//		IF(NOT simpleCommand.xError AND simpleCommand.xDone)THEN
//			iterateAndUpdateStatus.isInit := TRUE;
//			error := CRT_NO_ERROR;
//		END_IF
	CRT_CLOSE_COM_STATE:
		state := CRT_RESET_STATE;
		IF b_crt_close_enable THEN
			IF portOpened THEN
				crtClose(xExecute:=TRUE, hCom := openedHCom);
				IF crtClose.xError THEN
				   portOpened := FALSE;
				   crtClose.xExecute := FALSE;
				   state := CRT_INIT_STATE;
				   error := CRT_OPEN_ERROR;
				END_IF;
				IF crtClose.xDone THEN
					portOpened := FALSE;
				   crtClose.xExecute := FALSE;
				   state := CRT_INIT_STATE;
				END_IF;
			ELSE
				   state := CRT_INIT_STATE;
			END_IF
			
		END_IF
		
	
	CRT_STATUS_REQUEST_STATE:	
		simpleCommand(xExecute:=TRUE, hCom := openedHCom, xCommandDataSize:=0, xCommand:= CRT_STATUS_REQUEST_COMMAND , xCommandDataSize:=0);
		IF simpleCommand.xDone THEN
			newCardState := crtDecodeCardState(iST0:=simpleCommand.xST0, iST1:=simpleCommand.xST1);
			locked := (simpleCommand.xST1 = 16#30); 
			state := CRT_STATUS_REQUEST_STATE;
			waitTimer(IN:= TRUE, PT := POLL_DELAY);
			
		END_IF
		

		IF simpleCommand.xError THEN    
			newCardState := CRT_CARD_UNDEFINED;
			IF simpleCommand.xTimeout THEN
				state := CRT_CLOSE_COM_STATE;
				waitTimer(IN:= TRUE, PT := POLL_DELAY);
			ELSE
				//state := CRT_STATUS_REQUEST_STATE;
				state := CRT_CLOSE_COM_STATE;
				waitTimer(IN:= TRUE, PT := POLL_DELAY);
			END_IF
		END_IF	
	CRT_RF_CARD_RESET:
		simpleCommand(xExecute:=TRUE, hCom := openedHCom,  xCommand:= CRT_RF_CARD_RESET_COMMAND , 
				     xCommandDataSize:=UINT_TO_BYTE(SIZEOF(CRT_RF_CARD_RESET_COMMAND_DATA)), xCommandData := ADR (CRT_RF_CARD_RESET_COMMAND_DATA)) ;
		IF simpleCommand.xDone THEN
			//newCardState := crtDecodeCardState(iST0:=simpleCommand.xST0, iST1:=simpleCommand.xST1);
			newCardState :=CRT_RF_CARD_INSIDE;
			state := CRT_STATUS_REQUEST_STATE;
			waitTimer(IN:= TRUE, PT := POLL_DELAY);
			cardIdLen := simpleCommand.xOutputData[3];
			MEM.MemMove(pSource:=simpleCommand.xOutputData + 4, pDestination:=ADR(cardId), uiNumberOfBytes := MIN(cardIdLen, SIZEOF(cardId)));
			
		END_IF
		

		IF simpleCommand.xError THEN    
			newCardState := CRT_CARD_UNDEFINED;
			IF simpleCommand.xTimeout THEN
				//state := CRT_RESET_STATE;
				state := CRT_CLOSE_COM_STATE;
				waitTimer(IN:= TRUE, PT := POLL_DELAY);
			ELSE
				//state := CRT_STATUS_REQUEST_STATE;
				state := CRT_CLOSE_COM_STATE;
				waitTimer(IN:= TRUE, PT := POLL_DELAY);
			END_IF
		END_IF	

	CRT_LOCK:
		simpleCommand(xExecute:=TRUE, hCom := openedHCom, xCommandDataSize:=0, xCommand:= CRT_LATCH_LOCK_COMMAND , xCommandDataSize:=0);
		IF simpleCommand.xDone THEN
			newCardState := crtDecodeCardState(iST0:=simpleCommand.xST0, iST1:=simpleCommand.xST1);
			locked := (simpleCommand.xST1 = 16#30); 
			state := CRT_STATUS_REQUEST_STATE;
			waitTimer(IN:= TRUE, PT := POLL_DELAY);
			
		END_IF

		IF simpleCommand.xError THEN    
			newCardState := CRT_CARD_UNDEFINED;
			IF simpleCommand.xTimeout THEN
				//state := CRT_RESET_STATE;
				state := CRT_CLOSE_COM_STATE;
				waitTimer(IN:= TRUE, PT := POLL_DELAY);
			ELSE
				//state := CRT_STATUS_REQUEST_STATE;
				state := CRT_CLOSE_COM_STATE;
				waitTimer(IN:= TRUE, PT := POLL_DELAY);
			END_IF
		END_IF		

	CRT_RELEASE:
		simpleCommand(xExecute:=TRUE, hCom := openedHCom, xCommandDataSize:=0, xCommand:= CRT_LATCH_RELEASE_COMMAND , xCommandDataSize:=0);
		IF simpleCommand.xDone THEN
			newCardState := crtDecodeCardState(iST0:=simpleCommand.xST0, iST1:=simpleCommand.xST1);
			locked := (simpleCommand.xST1 = 16#30); 
			state := CRT_STATUS_REQUEST_STATE;
			waitTimer(IN:= TRUE, PT := POLL_DELAY);
			
		END_IF

		IF simpleCommand.xError THEN    
			newCardState := CRT_CARD_UNDEFINED;
			IF simpleCommand.xTimeout THEN
				//state := CRT_RESET_STATE;
				state := CRT_CLOSE_COM_STATE;
				waitTimer(IN:= TRUE, PT := POLL_DELAY);
			ELSE
				//state := CRT_STATUS_REQUEST_STATE;
				state := CRT_CLOSE_COM_STATE;
				waitTimer(IN:= TRUE, PT := POLL_DELAY);
			END_IF
		END_IF					
	
		
    CRT_FATAL_ERROR:
		state := CRT_CLOSE_COM_STATE;
	
//	CRT_DONE:  //all work is done, free resources
//		crtOpen(xExecute := FALSE);
//		state := CRT_DO_NOTHING;
//						
//	CRT_DO_NOTHING:
END_CASE

IF newCardState = CRT_CARD_INSIDE AND lastCardState = CRT_RF_CARD_INSIDE THEN 
	newCardState := CRT_RF_CARD_INSIDE;
END_IF

IF newCardState = CRT_CARD_INSIDE AND lastCardState <> CRT_CARD_INSIDE THEN
	//moment of inserting card
	state := CRT_RF_CARD_RESET;
	waitTimer(IN:= TRUE, PT := POLL_DELAY);
ELSIF newCardState <> CRT_CARD_INSIDE AND newCardState <> CRT_RF_CARD_INSIDE THEN
	cardIdLen :=0; //reset card id
	
END_IF		
lastCardState := newCardState;

iterateAndUpdateStatus.cardState := newCardState;
iterateAndUpdateStatus.busy := simpleCommand.xExecute OR NOT crtOpen.xDone;
//iterateAndUpdateStatus.busy := (simpleCommand.xExecute AND NOT simpleCommand.xDone) OR NOT crtOpen.xDone;
iterateAndUpdateStatus.locked := locked;
iterateAndUpdateStatus.error := error;
END_METHOD

METHOD latchLock
//very stupid
IF  state <> CRT_FATAL_ERROR AND state <> CRT_DONE AND state <> CRT_RESET_STATE AND state<>CRT_DO_NOTHING THEN
	state:= CRT_LOCK;

END_IF
END_METHOD

METHOD latchRelease
IF  state <> CRT_FATAL_ERROR AND state <> CRT_DONE AND state <> CRT_RESET_STATE AND state<>CRT_DO_NOTHING THEN
	state:= CRT_RELEASE;

END_IF
END_METHOD

END_FUNCTION_BLOCK

// CompWin/AppTerminalPost/DevCard/crtSimpleCommand
///command 
FUNCTION_BLOCK crtSimpleCommand
VAR CONSTANT
	STATE_INITIAL: BYTE := 0;
	STATE_WAIT_ACK: BYTE := 1;
	STATE_FATAL_ERROR: BYTE := 3;
	STATE_WAIT_RESPONSE: BYTE := 4;
	STATE_SEND_ACK: BYTE := 5;
	///minimal answer
	COMMAND_MINIMAL_ANSWER_SIZE: BYTE := 9;
	///maximum size of command data 
	COMMAND_DATA_SIZE_MAX: BYTE := 5;
	///maximum size of response 
	RESPONSE_DATA_SIZE_MAX: BYTE := 255;
	COMMAND_DATA_OFFSET: BYTE := 6;
	RESPONSE_DATA_OFFSET: BYTE := 8;
	ACK: BYTE := 16#6;
	///? 
	TIMEOUT: TIME := TIME#2s0ms;
END_VAR
VAR_INPUT
	hCom: CAA.HANDLE;
	xExecute: BOOL := FALSE;
	///device address
	xDestinationId: BYTE := 2;
	///master address, default = 1;
	xSourceId: BYTE := 1;
	xCommand: crtParametrizedCommand;
	xCommandData: POINTER TO BYTE;
	xCommandDataSize: BYTE := 0;
END_VAR
VAR_OUTPUT
	xDone: BOOL := FALSE;
	xError: BOOL := FALSE;
	xTimeout: BOOL := FALSE;
	///status characters
	xST0: BYTE;
	xST1: BYTE;
	///error codes
	xE0: BYTE;
	xE1: BYTE;
	xOutputData: POINTER TO BYTE := ((ADR(readBuffer) + RESPONSE_DATA_OFFSET) + 1);
	xOutputDataSize: BYTE;
END_VAR
VAR
	///buffer for command
	commandBuffer: ARRAY[0..(((2 + 3) + COMMAND_DATA_SIZE_MAX) + 2)] OF BYTE;
	///size enough for ack and answer
	readBuffer: ARRAY[0..(((3 + 3) + RESPONSE_DATA_SIZE_MAX) + 2)] OF BYTE;
	///timeout timer (timeout value - ????)
	waitingACKtimeout: TON;
	localState: BYTE := STATE_INITIAL;
	crtCOMWrite: COM.Write;
	crtCOMRead: COM.Read;
	bufferReaded: CAA.SIZE := 0;
	bufferFullLen: BYTE := 5;
	///full answer size with echo
	fullAnswerSize: BYTE;
	errorExecuting: BOOL;
	commandCode: INT;
	bcc: BYTE;
END_VAR

CASE localState OF 
	STATE_INITIAL:
		IF xExecute THEN
			xDone := FALSE;
			xError := FALSE;
			xTimeout := FALSE;
			IF NOT crtCOMWrite.xExecute THEN //at first time fill buffer
				bufferFullLen := 3 + 3 + xCommandDataSize + 2;  
				commandBuffer[0] := 16#F2;    //header 1
				commandBuffer[1] := 0;    //data len msb
				commandBuffer[2] := 3 + xCommandDataSize; //data len lsb
				commandBuffer[3] := 16#43;
				commandBuffer[4] := xCommand.CM; 		   //CM (command character)
				commandBuffer[5] := xCommand.PM;  //PM (parameter character)
				xOutputDataSize := 0;
				IF xCommandDataSize > 0 THEN
					MEM.MemMove(pSource := xCommandData, pDestination := ADR(commandBuffer) + COMMAND_DATA_OFFSET, uiNumberOfBytes := xCommandDataSize);
				END_IF;
				commandBuffer[6 + xCommandDataSize]:= 3; //don't know, what is it
				commandBuffer[7 + xCommandDataSize] := crtBCC(iCommandBuffer := ADR(commandBuffer) , iCommandBufferSize := bufferFullLen);
				xE0 :=0;
				xE1 :=0;
				errorExecuting :=FALSE;

			END_IF
			crtCOMWrite(xExecute := TRUE,hCom:= hCom, pBuffer:= ADR(commandBuffer), szSize:= bufferFullLen);
			IF crtCOMWrite.xError THEN
				xError := TRUE;
				xExecute := FALSE;
				xCommandDataSize :=0;
				localState := STATE_INITIAL;
				crtCOMWrite(xExecute := FALSE);
				RETURN;
			END_IF
		
			// if the writing process is completed the reading process can be started
			IF crtCOMWrite.xDone THEN
				localState := STATE_WAIT_RESPONSE;
				bufferReaded := 0;
				xCommandDataSize :=0;
				crtCOMWrite(xExecute := FALSE);
				fullAnswerSize := COMMAND_MINIMAL_ANSWER_SIZE; //wait for ack + response
				errorExecuting := FALSE;
				waitingACKtimeout(IN:=FALSE); 
				waitingACKtimeout(IN:=TRUE, PT:=TIMEOUT);  //timeout value ?
			END_IF			
		END_IF
	//waiting response and ack
	STATE_WAIT_RESPONSE:
		waitingACKtimeout(IN:=TRUE, PT:=TIMEOUT);  //timeout value ?
		IF waitingACKTimeout.Q THEN  //timeout is over..
			xError := TRUE;
			xExecute := FALSE;
			xTimeout := TRUE;
			localState := STATE_INITIAL;
			crtCOMRead(xExecute := FALSE);
		ELSE
			crtCOMRead(xExecute := FALSE);
			crtCOMRead(xExecute := TRUE,hCom:= hCom, pBuffer:= ADR(readBuffer) + bufferReaded, szBuffer:= SIZEOF(readBuffer) - bufferReaded);
			IF crtCOMRead.xError THEN
				xError := TRUE;
				xExecute := FALSE;
				crtCOMRead(xExecute := FALSE);
				localState := STATE_INITIAL;
			END_IF
			//After completion the size of the written bytes are saved
			IF 	crtCOMRead.xDone THEN
				bufferReaded := bufferReaded + crtCOMRead.szSize;
				//if first byte not ack-errir
				IF bufferReaded >=1 AND readBuffer[0]<> ACK THEN
					xError := TRUE;
					xExecute := FALSE;
					crtCOMRead(xExecute := FALSE);
					localState := STATE_INITIAL;
					RETURN;
				END_IF 
				IF bufferReaded >= fullAnswerSize THEN  //try to recognize command
					crtCOMRead(xExecute := FALSE);
					//ALL OK
					IF (readBuffer[1] = 16#F2 AND readBuffer[5]= xCommand.CM AND readBuffer[6]= xCommand.PM ) THEN  //receive response
						localState := STATE_WAIT_RESPONSE;
						fullAnswerSize := readBuffer[3] + 5 + 1; //extract response data size from readbuffer (with ACK FIRST BYTE)
						IF (bufferReaded >= fullAnswerSize ) THEN
							crtCOMRead(xExecute := FALSE);
							bcc := crtBCC(iCommandBuffer := ADR(readBuffer) +1, iCommandBufferSize := fullAnswerSize-1);
							IF bcc = readBuffer[fullAnswerSize - 1] AND readBuffer[4] = 16#50 THEN  //ordinary response, all ok
								xST1:= readBuffer[7];
								xST0:= readBuffer[8];
								xOutputDataSize := readBuffer[3] - 3;
								localState := STATE_SEND_ACK;
							ELSIF bcc = readBuffer[fullAnswerSize - 1] AND readBuffer[4] = 16#4E THEN //irregular response 								
								xE1:=readBuffer[7];
								xE0:=readBuffer[8];
								xOutputDataSize := readBuffer[3] - 3;
								errorExecuting := TRUE;
								localState := STATE_SEND_ACK;
							ELSE
								xError := TRUE;
								xExecute := FALSE;
								localState := STATE_INITIAL;
							END_IF
						END_IF
					ELSE
						xError := TRUE;
						xExecute := FALSE;
						localState := STATE_INITIAL;
					END_IF
				END_IF

			END_IF			
		END_IF
	STATE_SEND_ACK:
		commandBuffer[0] := 16#06; //ACK 
		crtCOMWrite(xExecute := TRUE,hCom:= hCom, pBuffer:= ADR(commandBuffer), szSize:= 1); //send ack
		IF crtCOMWrite.xError OR crtCOMWrite.xDone  THEN
				xExecute := FALSE;
				xError := errorExecuting;
				xDone := NOT (xError);
				
				xCommandDataSize :=0;
				localState := STATE_INITIAL;
				crtCOMWrite(xExecute := FALSE);
				RETURN;
		END_IF
		
		
		
END_CASE

END_FUNCTION_BLOCK

// CompWin/AppTerminalPost/DevCard/crtBCC
///calculate BCC (exclusive-or-verify) for buffer; receive full command buffer
FUNCTION crtBCC : BYTE
VAR_INPUT
	iCommandBuffer: POINTER TO BYTE;
	iCommandBufferSize: WORD;
END_VAR
VAR
	i: WORD;
END_VAR

crtBCC := 0;
FOR i := 0 TO iCommandBufferSize - 2 DO
	crtBCC := crtBCC XOR iCommandBuffer[i];
END_FOR

END_FUNCTION

// CompWin/AppTerminalPost/DevCard/crtDecodeCardState
///process ST0 and ST1 status command output
FUNCTION crtDecodeCardState : CRT_CARD_STATE
VAR_INPUT
	iST0: BYTE;
	iST1: BYTE;
END_VAR

crtDecodeCardState := CRT_CARD_UNDEFINED;
IF (iST0 =16#30 OR iST0 = 16#31) THEN
	crtDecodeCardState := CRT_NO_CARD;
ELSIF iST0 = 16#32 THEN
	crtDecodeCardState := CRT_CARD_INSIDE;
END_IF

END_FUNCTION

// CompWin/AppTerminalPost/StdLogger
FUNCTION_BLOCK StdLogger
VAR_INPUT
	sCmpName  : STRING;
END_VAR
VAR_OUTPUT
END_VAR
VAR
	udiCmpId : UDINT;
	udiCmpVersion : UDINT;
	vendorId : UDINT := 16#11110000;
	cmpId : UDINT := 16#0123;
	hCmp : RTS_IEC_HANDLE;
	hStdLogger : RTS_IEC_HANDLE;
	Result : RTS_IEC_RESULT;
	c: INT := 0;	
END_VAR

udiCmpId := vendorId OR Component_Manager.ComponentID.CMPID_IecCode OR cmpId;
udiCmpVersion := 16#03050000;
//sCmpName := 'CashCode';
//hCmp := CMAddComponent(sCmpName, udiCmpId, udiCmpVersion, ADR(Result)); 
hCmp := CMAddComponent('CashCode', udiCmpId, udiCmpVersion, ADR(Result));

METHOD AddLogEntry : BOOL
VAR_INPUT
	udiClassId : UDINT;
	sText : WSTRING;
END_VAR
VAR
	str: STRING;
	udiErrorId : UDINT := Errors.ERR_FAILED;
	udiInfoId : UDINT := 0;
END_VAR
AddLogEntry := FALSE;
str := WSTRING_TO_STRING(sText);
IF (LogAdd2(hStdLogger, udiCmpId, udiClassId, udiErrorId, udiInfoId, str) = Errors.ERR_OK) THEN
	AddLogEntry := TRUE;
END_IF;
END_METHOD

METHOD debug
VAR_INPUT
	msg: WSTRING;
END_VAR
AddLogEntry(CmpLog.LogClass.LOG_DEBUG, msg);
END_METHOD

METHOD error
VAR_INPUT
	msg: WSTRING;
END_VAR
AddLogEntry(CmpLog.LogClass.LOG_ERROR, msg);
END_METHOD

METHOD FB_Exit : BOOL
VAR_INPUT
	bInCopyCode : BOOL;  // if TRUE, the instance afterwards gets moved into the copy code (online change)	
END_VAR
CMRemoveComponent(hCmp);
FB_exit := TRUE;
END_METHOD

METHOD FB_Init : BOOL
VAR_INPUT
	bInitRetains : BOOL; // if TRUE, the retain variables are initialized (warm start / cold start)
	bInCopyCode : BOOL;  // if TRUE, the instance afterwards gets moved into the copy code (online change)	
END_VAR
c := c + 1;

hStdLogger := LogOpen('PlcLog', 0);
FB_Init := TRUE;
END_METHOD

METHOD info
VAR_INPUT
	msg: WSTRING;
END_VAR
AddLogEntry(CmpLog.LogClass.LOG_INFO, msg);
END_METHOD

METHOD warn
VAR_INPUT
	msg: WSTRING;
END_VAR
AddLogEntry(CmpLog.LogClass.LOG_WARNING, msg);
END_METHOD

END_FUNCTION_BLOCK

// CompWin/AppTerminalPost/Post/SafePrg
PROGRAM SafePrg

// сохранить retain в файл
IF(RetainManager.Init)THEN
//	RetainManager(ForceRestore := FALSE, ForceSave := TRUE, ForceBalance := FALSE);
	RetainManager(ForceRestore := FALSE, ForceSave := FALSE, ForceBalance := FALSE);
END_IF

END_PROGRAM

// CompWin/AppTerminalPost/Traffic/DataToSpk
PROGRAM DataToSpk
VAR
	_activeButton : INT;
END_VAR

// номер поста
//go_postNumber := PLC_PRG.post.Number;
// выбранная функция
_activeButton := DeviceButtons.GetActiveButton();// PLC_PRG.post.Mode;
// для режимов не_мойки не передавать ничего в Контроллер
//IF(PLC_PRG.post.Mode = EnumMode.CASHCOLLECT)THEN
IF(NOT PLC_PRG.post.IsReadyToWash())THEN
	spk_data.go_postFunction := EnumButton.NONE;
ELSE
	spk_data.go_postFunction := _activeButton;
END_IF


// изменение для замены местами пены и шампуня
IF(spk_data.go_postFunction = 2)THEN
	spk_data.go_postFunction := 3;
ELSIF(spk_data.go_postFunction = 3)THEN
	spk_data.go_postFunction := 2;
END_IF

// баланс поста
spk_data.go_postCounterFund := REAL_TO_INT(PLC_PRG.post.CounterFund);

// счётчики банкнот
SPK_DATA.counterBanknote10 := DeviceBanknote.GetCounterBanknote(10);
SPK_DATA.counterBanknote50 := DeviceBanknote.GetCounterBanknote(50);
SPK_DATA.counterBanknote100 := DeviceBanknote.GetCounterBanknote(100);
SPK_DATA.counterBanknote500 := DeviceBanknote.GetCounterBanknote(500);
SPK_DATA.counterBanknote1000 := DeviceBanknote.GetCounterBanknote(1000);
SPK_DATA.counterBanknote5000 := DeviceBanknote.GetCounterBanknote(5000);

// счётчики монет
SPK_DATA.counterCoin := DeviceCoin.GetCounterCoin(0);
SPK_DATA.counterCoin1 := DeviceCoin.GetCounterCoin(1);
SPK_DATA.counterCoin2 := DeviceCoin.GetCounterCoin(2);
SPK_DATA.counterCoin5 := DeviceCoin.GetCounterCoin(5);
SPK_DATA.counterCoin10 := DeviceCoin.GetCounterCoin(10);

SPK_DATA.fundFromCollect := PLC_PRG.post.GeFundFromCollect();
SPK_DATA.fundTotal := PLC_PRG.post.GetFundTotal();

// сообщения
SPK_DATA.messageInCash := PLC_PRG.post.GetMessageInCash();
SPK_DATA.messageFunc := PLC_PRG.post.GetMessageFunc();
SPK_DATA.messageCollect := PLC_PRG.post.GetMessageCollect();
SPK_DATA.messageTotal := PLC_PRG.post.GetMessageTotal();

// счетчик для контроля связи и работы терминала
spk_data.go_counter := spk_data.go_counter + 1;

// показать текущие тарифы мойки
SPK_DATA.currentRates[0] := PersistentVars.rates[0];
SPK_DATA.currentRates[1] := PersistentVars.rates[1];
SPK_DATA.currentRates[2] := PersistentVars.rates[2];
SPK_DATA.currentRates[3] := PersistentVars.rates[3];
SPK_DATA.currentRates[4] := PersistentVars.rates[4];
SPK_DATA.currentRates[5] := PersistentVars.rates[5];
SPK_DATA.currentRates[6] := PersistentVars.rates[6];
SPK_DATA.currentRates[7] := PersistentVars.rates[7];
SPK_DATA.currentRates[8] := PersistentVars.rates[8];


// Флаги купюрника
SPK_DATA.cashcodeStatus := DeviceBanknote.cashcodeStatus;
SPK_DATA.cashcodeError := DeviceBanknote.cashcodeError;
SPK_DATA.casetteDropped := DeviceBanknote.IsCasetteDropped();
SPK_DATA.banknoteJammed := DeviceBanknote.IsBanknoteJammed();

// Флаги блокировки дверей
// 1 - замок закрыт; 0 - замок открыт
IF(PLC_PRG.post.Locks[EnumLock.LOCK_TOP])THEN
	SPK_DATA.lockTop := 1;
ELSE
	SPK_DATA.lockTop := 0;
END_IF

// состояние среднего замка
IF(PLC_PRG.post.Locks[EnumLock.LOCK_MID])THEN
	SPK_DATA.lockMid := 1;
ELSE
	SPK_DATA.lockMid := 0;
END_IF

// текущие паузы режимов
SPK_DATA.currentPauseActiveClean := TIME_TO_WORD(PLC_PRG.post.GetPauseActiveClean() / 1000);
SPK_DATA.currentPauseFoam := TIME_TO_WORD(PLC_PRG.post.GetPauseFoam() / 1000);
SPK_DATA.currentPauseShampoo := TIME_TO_WORD(PLC_PRG.post.GetPauseShampoo() / 1000);

END_PROGRAM

// CompWin/AppTerminalPost/Traffic/DataToUI
PROGRAM DataToUI
VAR
END_VAR

// номер поста
NVL2UI.postNumber := PLC_PRG.post.Number;
	
// Состояние терминала: ожидание, функции, окончание мойки, уборка, инкассация, пополнение баланса оператором
NVL2UI.postMode := PLC_PRG.post.Mode;
IF(PLC_PRG.post.ActiveCardType = EnumCardType.CLEANUP)THEN
	NVL2UI.postMode := EnumMode.CLEANUP;
//ELSIF(PLC_PRG.post.ActiveCardType = EnumCardType.CASHCOLLECT)THEN
//	
END_IF

// Для REAL отбросываю дробную часть DINT_TO_INT(TRUNC(real));
// REAL_TO_WORD(real);	// округление до ближайшего целого
// баланс
NVL2UI.postCounterFund := DINT_TO_INT(TRUNC(PLC_PRG.post.CounterFund));

// тип карты
NVL2UI.cardType := PLC_PRG.post.ActiveCardType;

	
// нажатая кнопка
NVL2UI.buttonActive := DeviceButtons.GetActiveButton();
// изменение для замены местами пены и шампуня
IF(NVL2UI.buttonActive = 2)THEN
	NVL2UI.buttonActive := 3;
ELSIF(NVL2UI.buttonActive = 3)THEN
	NVL2UI.buttonActive := 2;
END_IF
		
// сумма внесения
NVL2UI.amountReceived := WORD_TO_INT(PLC_PRG.post.Received);
	
IF(PLC_PRG.post.FinCostSummary <> '')THEN	
	// внесено за мойку
	//NVL2UI.paidWash := PLC_PRG.post.InCash;
	// стоимость оконченной мойки
	NVL2UI.costWash := DINT_TO_INT(TRUNC(PLC_PRG.post.costWash));
	// сдача
	NVL2UI.costChange := 0;//DINT_TO_INT(TRUNC(PLC_PRG.post.InCash - PLC_PRG.post.costWash));
	// стоимость активной химии
	NVL2UI.costActiveClean := DINT_TO_INT(TRUNC(PLC_PRG.post.ModesLog[EnumMode.ACTIVECLEAN].Cost));
	// стоимость пены
	NVL2UI.costFoam :=  DINT_TO_INT(TRUNC(PLC_PRG.post.ModesLog[EnumMode.FOAM].Cost));
	// стоимость шампуня
	NVL2UI.costShampoo :=  DINT_TO_INT(TRUNC(PLC_PRG.post.ModesLog[EnumMode.SHAMPOO].Cost));
	// стоимость ХВ
	NVL2UI.costColdWater :=  DINT_TO_INT(TRUNC(PLC_PRG.post.ModesLog[EnumMode.COLDWATER].Cost));
	// стоимость ГВ
	NVL2UI.costHotWater :=  DINT_TO_INT(TRUNC(PLC_PRG.post.ModesLog[EnumMode.HOTWATER].Cost));
	// стоимость воска
	NVL2UI.costWax :=  DINT_TO_INT(TRUNC(PLC_PRG.post.ModesLog[EnumMode.WAX].Cost));
	// стоимость осмоса
	NVL2UI.costOsmose :=  DINT_TO_INT(TRUNC(PLC_PRG.post.ModesLog[EnumMode.OSMOSE].Cost));
	// стоимость паузы
	NVL2UI.costPause :=  DINT_TO_INT(TRUNC(PLC_PRG.post.ModesLog[EnumMode.PAUSE].Cost));
ELSE
	// стоимость оконченной мойки
	NVL2UI.costWash := 0;
	// сдача
	NVL2UI.costChange := 0;
	// стоимость активной химии
	NVL2UI.costActiveClean := 0;
	// стоимость пены
	NVL2UI.costFoam := 0;
	// стоимость шампуня
	NVL2UI.costShampoo := 0;
	// стоимость ХВ
	NVL2UI.costColdWater := 0;
	// стоимость ГВ
	NVL2UI.costHotWater := 0;
	// стоимость воска
	NVL2UI.costWax := 0;
	// стоимость осмоса
	NVL2UI.costOsmose := 0;
	// стоимость паузы
	NVL2UI.costPause := 0;
END_IF

	
// состояние верхнего замка
// 1 - замок закрыт; 0 - замок открыт
IF(PLC_PRG.post.Locks[EnumLock.LOCK_TOP])THEN
	NVL2UI.lockTop := 1;
ELSE
	NVL2UI.lockTop := 0;
END_IF

// состояние среднего замка
IF(PLC_PRG.post.Locks[EnumLock.LOCK_MID])THEN
	NVL2UI.lockMid := 1;
ELSE
	NVL2UI.lockMid := 0;
END_IF

END_PROGRAM

// CompWin/AppTerminalPost/DevCard/Cards
FUNCTION_BLOCK PUBLIC Cards
VAR_INPUT
END_VAR
VAR_OUTPUT
END_VAR
VAR
	rAmountOflock:			REAL;	//Максимальная сумма блокировки по карте (руб)
	uUnspentFundsID:		UINT;	//Карта (счёт) неиспользованных средств ()
END_VAR

END_FUNCTION_BLOCK

// CompWin/AppTerminalPost/DevCoin/ccTalkGetNoDataCommandBuffer
///create command buffer with no data for CCTALK
FUNCTION ccTalkGetNoDataCommandBuffer : ARRAY[0..4] OF BYTE
VAR CONSTANT
	BUFFER_SIZE: BYTE := 5;
END_VAR
VAR_INPUT
	iDestination: BYTE := 2;
	iCommandCode: BYTE;
	iSource: BYTE := 1;
END_VAR
VAR
	crc: BYTE;
END_VAR

ccTalkGetNoDataCommandBuffer[0] := iDestination;
ccTalkGetNoDataCommandBuffer[1] := 0; //data size 
ccTalkGetNoDataCommandBuffer[2] := iSource;  // master address
ccTalkGetNoDataCommandBuffer[3] := iCommandCode; //command code
ccTalkGetNoDataCommandBuffer[4] := ccTalkCRC(ADR(ccTalkGetNoDataCommandBuffer), SIZEOF(ccTalkGetNoDataCommandBuffer)); //command code

{
crc:=cacheCodeCrc(iCommandBuffer := ADR(cacheCodeGetNoDataCommandBuffer), iCommandBufferSize := BUFFER_SIZE);
cacheCodeGetNoDataCommandBuffer[4] := WORD_TO_BYTE(crc); //LSB FIrst
cacheCodeGetNoDataCommandBuffer[5] := WORD_TO_BYTE(SHR(crc, 8));
}

END_FUNCTION

// CompWin/AppTerminalPost/DevCard/crtInitCommand
FUNCTION_BLOCK crtInitCommand EXTENDS crtSimpleCommand

END_FUNCTION_BLOCK

// CompWin/AppTerminalPost/DevPrinter/unicode2cp866
FUNCTION unicode2cp866 : STRING(255)
VAR_INPUT
	str: WSTRING(255);
END_VAR
VAR
	i: INT;
	char: UINT;
	cp866char: USINT;
END_VAR

unicode2cp866:='';
FOR i:=0 TO WLEN(str)-1 DO
	char:= str[i];
	CASE char OF
		16#0 : cp866char:=16#0;
		16#1 : cp866char:=16#1;
		16#2 : cp866char:=16#2;
		16#3 : cp866char:=16#3;
		16#4 : cp866char:=16#4;
		16#5 : cp866char:=16#5;
		16#6 : cp866char:=16#6;
		16#7 : cp866char:=16#7;
		16#8 : cp866char:=16#8;
		16#9 : cp866char:=16#9;
		16#A : cp866char:=16#A;
		16#B : cp866char:=16#B;
		16#C : cp866char:=16#C;
		16#D : cp866char:=16#D;
		16#E : cp866char:=16#E;
		16#F : cp866char:=16#F;
		16#10 : cp866char:=16#10;
		16#11 : cp866char:=16#11;
		16#12 : cp866char:=16#12;
		16#13 : cp866char:=16#13;
		16#14 : cp866char:=16#14;
		16#15 : cp866char:=16#15;
		16#16 : cp866char:=16#16;
		16#17 : cp866char:=16#17;
		16#18 : cp866char:=16#18;
		16#19 : cp866char:=16#19;
		16#1A : cp866char:=16#1A;
		16#1B : cp866char:=16#1B;
		16#1C : cp866char:=16#1C;
		16#1D : cp866char:=16#1D;
		16#1E : cp866char:=16#1E;
		16#1F : cp866char:=16#1F;
		16#20 : cp866char:=16#20;
		16#21 : cp866char:=16#21;
		16#22 : cp866char:=16#22;
		16#23 : cp866char:=16#23;
		16#24 : cp866char:=16#24;
		16#25 : cp866char:=16#25;
		16#26 : cp866char:=16#26;
		16#27 : cp866char:=16#27;
		16#28 : cp866char:=16#28;
		16#29 : cp866char:=16#29;
		16#2A : cp866char:=16#2A;
		16#2B : cp866char:=16#2B;
		16#2C : cp866char:=16#2C;
		16#2D : cp866char:=16#2D;
		16#2E : cp866char:=16#2E;
		16#2F : cp866char:=16#2F;
		16#30 : cp866char:=16#30;
		16#31 : cp866char:=16#31;
		16#32 : cp866char:=16#32;
		16#33 : cp866char:=16#33;
		16#34 : cp866char:=16#34;
		16#35 : cp866char:=16#35;
		16#36 : cp866char:=16#36;
		16#37 : cp866char:=16#37;
		16#38 : cp866char:=16#38;
		16#39 : cp866char:=16#39;
		16#3A : cp866char:=16#3A;
		16#3B : cp866char:=16#3B;
		16#3C : cp866char:=16#3C;
		16#3D : cp866char:=16#3D;
		16#3E : cp866char:=16#3E;
		16#3F : cp866char:=16#3F;
		16#40 : cp866char:=16#40;
		16#41 : cp866char:=16#41;
		16#42 : cp866char:=16#42;
		16#43 : cp866char:=16#43;
		16#44 : cp866char:=16#44;
		16#45 : cp866char:=16#45;
		16#46 : cp866char:=16#46;
		16#47 : cp866char:=16#47;
		16#48 : cp866char:=16#48;
		16#49 : cp866char:=16#49;
		16#4A : cp866char:=16#4A;
		16#4B : cp866char:=16#4B;
		16#4C : cp866char:=16#4C;
		16#4D : cp866char:=16#4D;
		16#4E : cp866char:=16#4E;
		16#4F : cp866char:=16#4F;
		16#50 : cp866char:=16#50;
		16#51 : cp866char:=16#51;
		16#52 : cp866char:=16#52;
		16#53 : cp866char:=16#53;
		16#54 : cp866char:=16#54;
		16#55 : cp866char:=16#55;
		16#56 : cp866char:=16#56;
		16#57 : cp866char:=16#57;
		16#58 : cp866char:=16#58;
		16#59 : cp866char:=16#59;
		16#5A : cp866char:=16#5A;
		16#5B : cp866char:=16#5B;
		16#5C : cp866char:=16#5C;
		16#5D : cp866char:=16#5D;
		16#5E : cp866char:=16#5E;
		16#5F : cp866char:=16#5F;
		16#60 : cp866char:=16#60;
		16#61 : cp866char:=16#61;
		16#62 : cp866char:=16#62;
		16#63 : cp866char:=16#63;
		16#64 : cp866char:=16#64;
		16#65 : cp866char:=16#65;
		16#66 : cp866char:=16#66;
		16#67 : cp866char:=16#67;
		16#68 : cp866char:=16#68;
		16#69 : cp866char:=16#69;
		16#6A : cp866char:=16#6A;
		16#6B : cp866char:=16#6B;
		16#6C : cp866char:=16#6C;
		16#6D : cp866char:=16#6D;
		16#6E : cp866char:=16#6E;
		16#6F : cp866char:=16#6F;
		16#70 : cp866char:=16#70;
		16#71 : cp866char:=16#71;
		16#72 : cp866char:=16#72;
		16#73 : cp866char:=16#73;
		16#74 : cp866char:=16#74;
		16#75 : cp866char:=16#75;
		16#76 : cp866char:=16#76;
		16#77 : cp866char:=16#77;
		16#78 : cp866char:=16#78;
		16#79 : cp866char:=16#79;
		16#7A : cp866char:=16#7A;
		16#7B : cp866char:=16#7B;
		16#7C : cp866char:=16#7C;
		16#7D : cp866char:=16#7D;
		16#7E : cp866char:=16#7E;
		16#7F : cp866char:=16#7F;
		16#410 : cp866char:=16#80;
		16#411 : cp866char:=16#81;
		16#412 : cp866char:=16#82;
		16#413 : cp866char:=16#83;
		16#414 : cp866char:=16#84;
		16#415 : cp866char:=16#85;
		16#416 : cp866char:=16#86;
		16#417 : cp866char:=16#87;
		16#418 : cp866char:=16#88;
		16#419 : cp866char:=16#89;
		16#41A : cp866char:=16#8A;
		16#41B : cp866char:=16#8B;
		16#41C : cp866char:=16#8C;
		16#41D : cp866char:=16#8D;
		16#41E : cp866char:=16#8E;
		16#41F : cp866char:=16#8F;
		16#420 : cp866char:=16#90;
		16#421 : cp866char:=16#91;
		16#422 : cp866char:=16#92;
		16#423 : cp866char:=16#93;
		16#424 : cp866char:=16#94;
		16#425 : cp866char:=16#95;
		16#426 : cp866char:=16#96;
		16#427 : cp866char:=16#97;
		16#428 : cp866char:=16#98;
		16#429 : cp866char:=16#99;
		16#42A : cp866char:=16#9A;
		16#42B : cp866char:=16#9B;
		16#42C : cp866char:=16#9C;
		16#42D : cp866char:=16#9D;
		16#42E : cp866char:=16#9E;
		16#42F : cp866char:=16#9F;
		16#430 : cp866char:=16#A0;
		16#431 : cp866char:=16#A1;
		16#432 : cp866char:=16#A2;
		16#433 : cp866char:=16#A3;
		16#434 : cp866char:=16#A4;
		16#435 : cp866char:=16#A5;
		16#436 : cp866char:=16#A6;
		16#437 : cp866char:=16#A7;
		16#438 : cp866char:=16#A8;
		16#439 : cp866char:=16#A9;
		16#43A : cp866char:=16#AA;
		16#43B : cp866char:=16#AB;
		16#43C : cp866char:=16#AC;
		16#43D : cp866char:=16#AD;
		16#43E : cp866char:=16#AE;
		16#43F : cp866char:=16#AF;
		16#2591 : cp866char:=16#B0;
		16#2592 : cp866char:=16#B1;
		16#2593 : cp866char:=16#B2;
		16#2502 : cp866char:=16#B3;
		16#2524 : cp866char:=16#B4;
		16#2561 : cp866char:=16#B5;
		16#2562 : cp866char:=16#B6;
		16#2556 : cp866char:=16#B7;
		16#2555 : cp866char:=16#B8;
		16#2563 : cp866char:=16#B9;
		16#2551 : cp866char:=16#BA;
		16#2557 : cp866char:=16#BB;
		16#255D : cp866char:=16#BC;
		16#255C : cp866char:=16#BD;
		16#255B : cp866char:=16#BE;
		16#2510 : cp866char:=16#BF;
		16#2514 : cp866char:=16#C0;
		16#2534 : cp866char:=16#C1;
		16#252C : cp866char:=16#C2;
		16#251C : cp866char:=16#C3;
		16#2500 : cp866char:=16#C4;
		16#253C : cp866char:=16#C5;
		16#255E : cp866char:=16#C6;
		16#255F : cp866char:=16#C7;
		16#255A : cp866char:=16#C8;
		16#2554 : cp866char:=16#C9;
		16#2569 : cp866char:=16#CA;
		16#2566 : cp866char:=16#CB;
		16#2560 : cp866char:=16#CC;
		16#2550 : cp866char:=16#CD;
		16#256C : cp866char:=16#CE;
		16#2567 : cp866char:=16#CF;
		16#2568 : cp866char:=16#D0;
		16#2564 : cp866char:=16#D1;
		16#2565 : cp866char:=16#D2;
		16#2559 : cp866char:=16#D3;
		16#2558 : cp866char:=16#D4;
		16#2552 : cp866char:=16#D5;
		16#2553 : cp866char:=16#D6;
		16#256B : cp866char:=16#D7;
		16#256A : cp866char:=16#D8;
		16#2518 : cp866char:=16#D9;
		16#250C : cp866char:=16#DA;
		16#2588 : cp866char:=16#DB;
		16#2584 : cp866char:=16#DC;
		16#258C : cp866char:=16#DD;
		16#2590 : cp866char:=16#DE;
		16#2580 : cp866char:=16#DF;
		16#440 : cp866char:=16#E0;
		16#441 : cp866char:=16#E1;
		16#442 : cp866char:=16#E2;
		16#443 : cp866char:=16#E3;
		16#444 : cp866char:=16#E4;
		16#445 : cp866char:=16#E5;
		16#446 : cp866char:=16#E6;
		16#447 : cp866char:=16#E7;
		16#448 : cp866char:=16#E8;
		16#449 : cp866char:=16#E9;
		16#44A : cp866char:=16#EA;
		16#44B : cp866char:=16#EB;
		16#44C : cp866char:=16#EC;
		16#44D : cp866char:=16#ED;
		16#44E : cp866char:=16#EE;
		16#44F : cp866char:=16#EF;
		16#401 : cp866char:=16#F0;
		16#451 : cp866char:=16#F1;
		16#404 : cp866char:=16#F2;
		16#454 : cp866char:=16#F3;
		16#407 : cp866char:=16#F4;
		16#457 : cp866char:=16#F5;
		16#40E : cp866char:=16#F6;
		16#45E : cp866char:=16#F7;
		16#B0 : cp866char:=16#F8;
		16#2219 : cp866char:=16#F9;
		16#B7 : cp866char:=16#FA;
		16#221A : cp866char:=16#FB;
		16#2116 : cp866char:=16#FC;
		16#A4 : cp866char:=16#FD;
		16#25A0 : cp866char:=16#FE;
		16#A0 : cp866char:=16#FF;
		ELSE
			cp866char:=16#3F; //?

END_CASE	
	unicode2cp866 := CONCAT(unicode2cp866, USINT_TO_STRING(cp866char)); 	
END_FOR

END_FUNCTION
